FUNCTION_BLOCK FB_Lights
VAR_INPUT
END_VAR
VAR_OUTPUT
END_VAR
VAR
END_VAR

END_FUNCTION_BLOCK

(* stored: Version 1.1.0.1, ProductVersion 3.1.4024.11
   POU FB_Lights: Id {e9373f71-6e7d-4a04-865a-64e7b49a0a42}, SpecialFunc None *)
